FUNCTION_BLOCK AdsTcpUnitEx
VAR_INPUT
	setMode : INT(0..1);
END_VAR
VAR_OUTPUT
	bBusy : BOOL;
	err : BOOL;
	errid : UDINT;
END_VAR
VAR_OUTPUT
	areaSockets : ARRAY[1..6] OF POINTER TO AdsSocket; //only used for finding a socket by name
	subarea4Sockets : ARRAY[1..9] OF POINTER TO AdsSocket;
END_VAR
VAR
	socket : REFERENCE TO AdsSocket;
	
	transmissionQueue : AdsMessageQueue;
	nextTransmission : AdsMessage;
	
	mode : (SEND, QUEUE);
END_VAR

(*
this extended version of AdsTcp communication provides the option dynamically generates ADS messages into a queue
	due to the significant stack memory requirements, the QUEUE model can only be used on systems with adjustable stack
	
QUEUE mode:
	when a message is polled, a socket with the same recipient name is identified
		if the identified socket is ready to send, then the message is passed to the socket
		otherwise, the message is placed back into the queue
	if no socket with a matching name can be identified, then the message is discarded
	
SEND mode:
	sendMessage() specifies a recipient name and data contents
	if a socket matching the recipient name is identified and it is not busy or in error state, then the message is passed
*)

//areaSockets[1] := ADR(AREA_1);
//areaSockets[2] := ADR(AREA_2);
areaSockets[3] := ADR(AREA_3);
//areaSockets[4] := ADR(AREA_4);
//areaSockets[5] := ADR(AREA_5);
//areaSockets[6] := ADR(AREA_6);
(*
subarea4Sockets[1] := ADR(SUBAREA_4_1);
subarea4Sockets[2] := ADR(SUBAREA_4_2);
subarea4Sockets[3] := ADR(SUBAREA_4_3);
subarea4Sockets[4] := ADR(SUBAREA_4_4);
subarea4Sockets[5] := ADR(SUBAREA_4_5);
subarea4Sockets[6] := ADR(SUBAREA_4_6);
subarea4Sockets[7] := ADR(SUBAREA_4_7);
subarea4Sockets[8] := ADR(SUBAREA_4_8);
subarea4Sockets[9] := ADR(SUBAREA_4_9);
*)
blocks();

IF mode = QUEUE THEN
	pollAndSend();	
END_IF

METHOD PRIVATE blocks : BOOL
VAR_INPUT
END_VAR
(*
AREA_1(
	PrgName=> , 
	AmsNetId=> , 
	AmsPort=> , 
	receivingData=> , 
	sendingData=> , 
	readBusy=> , 
	readError=> , 
	readErrorId=> , 
	writeBusy=> , 
	writeError=> , 
	writeErrorId=> );

AREA_2(
	PrgName=> , 
	AmsNetId=> , 
	AmsPort=> , 
	receivingData=> , 
	sendingData=> , 
	readBusy=> , 
	readError=> , 
	readErrorId=> , 
	writeBusy=> , 
	writeError=> , 
	writeErrorId=> );
*)
AREA_3(
	PrgName=> , 
	AmsNetId=> , 
	AmsPort=> , 
	receivingData=> , 
	sendingData=> , 
	readBusy=> , 
	readError=> , 
	readErrorId=> , 
	writeBusy=> , 
	writeError=> , 
	writeErrorId=> );

(*
AREA_4(
	PrgName=> , 
	AmsNetId=> , 
	AmsPort=> , 
	receivingData=> , 
	sendingData=> , 
	readBusy=> , 
	readError=> , 
	readErrorId=> , 
	writeBusy=> , 
	writeError=> , 
	writeErrorId=> );
*)
(*
AREA_5(
	PrgName=> , 
	AmsNetId=> , 
	AmsPort=> , 
	receivingData=> , 
	sendingData=> , 
	readBusy=> , 
	readError=> , 
	readErrorId=> , 
	writeBusy=> , 
	writeError=> , 
	writeErrorId=> );
	
AREA_6(
	PrgName=> , 
	AmsNetId=> , 
	AmsPort=> , 
	receivingData=> , 
	sendingData=> , 
	readBusy=> , 
	readError=> , 
	readErrorId=> , 
	writeBusy=> , 
	writeError=> , 
	writeErrorId=> );
*)
END_METHOD

METHOD PRIVATE findSocket : REFERENCE TO AdsSocket
VAR_INPUT
	recipient : STRING;
END_VAR
VAR
	i : INT;
END_VAR
FOR i:=1 TO numSockets BY 1 DO
	IF areaSockets[i] <> 0 AND_THEN areaSockets[i]^.PrgName = recipient THEN
		findSocket REF= areaSockets[i]^;
		RETURN;
	END_IF
END_FOR

FOR i:=1 TO numSubarea4Sockets BY 1 DO
	IF subarea4Sockets[i] <> 0 AND_THEN subarea4Sockets[i]^.PrgName = recipient THEN
		findSocket REF= areaSockets[i]^;
		RETURN;
	END_IF
END_FOR
END_METHOD

METHOD PRIVATE pollAndSend : BOOL
VAR_INPUT
END_VAR
nextTransmission := transmissionQueue.poll(getSize => );
socket REF= findSocket(recipient := nextTransmission.recipient);

IF __ISVALIDREF(socket) THEN
	
	IF NOT socket.writeBusy AND NOT socket.writeError THEN
		socket.send(data := nextTransmission.contents);
	ELSE //if socket is busy or has ERROR state, then message is returned to the end of the line
		transmissionQueue.push(value := nextTransmission);
	END_IF
	
END_IF
END_METHOD

METHOD sendMessage : BOOL
VAR_INPUT
	recipient : STRING;
	data : REFERENCE TO AdsData;
END_VAR
VAR
	newMessage : AdsMessage;
END_VAR
CASE mode OF
	SEND:
		socket REF= findSocket(recipient := recipient);
		IF
			__ISVALIDREF(socket) AND_THEN
			NOT socket.writeBusy AND NOT socket.writeError
		THEN
			socket.send(data := data);
			sendMessage := TRUE;
		END_IF
	
	QUEUE:
		IF recipient <> '' THEN
			newMessage.recipient := recipient;
			newMessage.contents := data;
			
			sendMessage := transmissionQueue.push(newMessage);
		END_IF
	
END_CASE
END_METHOD

END_FUNCTION_BLOCK

(* stored: Version 1.1.0.1, ProductVersion 3.1.4024.11
   POU AdsTcpUnitEx: Id {fdbfe87f-1184-47dd-b08b-0750e1c8692f}, SpecialFunc None
   Method blocks: Id {84a4da9e-7305-47f8-b050-02c3484c700e}
   Method findSocket: Id {d8b3993d-426a-4e5d-a36f-587468829b99}
   Method pollAndSend: Id {018dc648-0b60-4c81-a6e8-f9e64516fdaa}
   Method sendMessage: Id {20b0f168-c0bb-48be-90d8-084d1d464586} *)
